(* PLC project KinIn_v3.project, CODESYS CODESYS V3.5 SP19 *)
(* stored: creationDateTime 2025-01-20T16:27:25.9240719, modificationDateTime 2025-01-20T16:17:39.6822999 *)

FUNCTION_BLOCK MatMul
  VAR_INPUT
    {attribute 'variable_length_array_original_scope' := 'Inout'}
    {attribute 'variable_length_array' := 'ARRAY[*,*] OF REAL'}
    {attribute 'Dimensions' := '2'}
    mat1 : POINTER TO REAL;
    {attribute 'variable_length_array_original_scope' := 'Inout'}
    {attribute 'variable_length_array' := 'ARRAY[*,*] OF REAL'}
    {attribute 'Dimensions' := '2'}
    mat2 : POINTER TO REAL;
    {attribute 'variable_length_array_original_scope' := 'Inout'}
    {attribute 'variable_length_array' := 'ARRAY[*,*] OF REAL'}
    {attribute 'Dimensions' := '2'}
    MatResult : POINTER TO REAL;
  END_VAR
  VAR
    i : DINT;
    j : DINT;
    k : DINT;
  END_VAR

            FOR i:=1 TO UPPER_BOUND(MatResult,1) DO
	FOR j:=1 TO UPPER_BOUND(MatResult,2) DO
		MatResult[i,j]:=0;
		FOR k:=1 TO UPPER_BOUND(mat2,1) DO//dimmension not appering in result
			MatResult[i,j]:=MatResult[i,j]+mat1[i,k]*mat2[k,j];
		END_FOR;
	END_FOR
END_FOR
          
END_FUNCTION_BLOCK
